# EPICS substitutions: devel/epics/drivers/jlabVMEBoardApp/Db/userHost.substitutions
# Example substitutions file

file "db/dbExample1.db" {
    { user = "hovanesHost" }
}

file db/dbExample2.db {
    pattern { user, no, scan }
        { "hovanesHost", 1, "1 second" }
        { "hovanesHost", 2, "2 second" }
        { "hovanesHost", 3, "5 second" }
}
